Fanuc KAREL source: GET_TIME.kl

PROGRAM T
%NOLOCKGROUP
VAR
 v0 : INTEGER
BEGIN
 GET_TIME(v0)
END T
